FUNCTION_BLOCK TwoConCtlMulticast (* Composite Function Block Type *)
  (* Standard: 61499-2 *)
  (* Version 0.2, 2003-12-05, JHC, Rockwell Automation, Renamed from NEWCOMPFB. *)
  (* Version 0.1, 2002-01-08, JHC, Rockwell Automation, Added DLY FB as example. *)
  (* Version 0.0, 2000-05-27, JHC, Rockwell Automation *)
  (* Compiler header: package fb.rt.cs725; *)
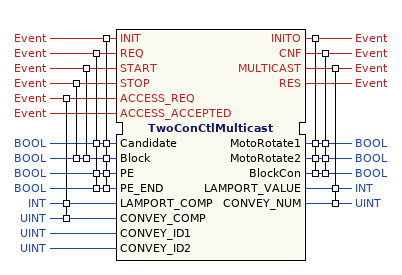
  EVENT_INPUT
    INIT WITH Candidate, Block, PE, PE_END; (* Initialization Request *)
    REQ WITH Candidate, PE, PE_END; (* Normal Execution Request *)
    START WITH Block;
    STOP WITH Block;
    ACCESS_REQ WITH LAMPORT_COMP, CONVEY_COMP;
    ACCESS_ACCEPTED;
  END_EVENT
  EVENT_OUTPUT
    INITO WITH MotoRotate1, MotoRotate2, BlockCon; (* Initialization Confirm *)
    CNF WITH MotoRotate1, MotoRotate2, BlockCon; (* Execution Confirmation *)
    MULTICAST WITH LAMPORT_VALUE, CONVEY_NUM;
    RES;
  END_EVENT
  VAR_INPUT
    Candidate : BOOL;
    Block : BOOL;
    PE : BOOL;
    PE_END : BOOL;
    LAMPORT_COMP : INT;
    CONVEY_COMP : UINT;
    CONVEY_ID1 : UINT;
    CONVEY_ID2 : UINT;
  END_VAR
  VAR_OUTPUT
    MotoRotate1 : BOOL;
    MotoRotate2 : BOOL;
    BlockCon : BOOL;
    LAMPORT_VALUE : INT;
    CONVEY_NUM : UINT;
  END_VAR
  FBS
    FC11 : ConveyorCTLMulticast(PE := 1, Block := 0, Candidate := 0);
    FC12 : ConveyorCTLMulticast;
  END_FBS
  EVENT_CONNECTIONS
    INIT TO FC11.INIT;
    REQ TO FC11.REQ;
    FC12.INITO TO INITO;
    FC12.CNF TO CNF;
    REQ TO FC12.REQ;
    STOP TO FC12.CAS_STOP;
    START TO FC12.CAS_START;
    FC12.STOP TO FC11.CAS_STOP;
    FC12.START TO FC11.CAS_START;
    FC11.INITO TO FC12.INIT;
    FC12.MULTICAST TO MULTICAST;
    FC12.RES TO RES;
    ACCESS_REQ TO FC12.ACCESS_REQ;
    ACCESS_ACCEPTED TO FC12.ACCESS_ACCEPTED;
  END_CONNECTIONS
  DATA_CONNECTIONS
    Block TO FC12.Block;
    Candidate TO FC12.Candidate;
    PE TO FC12.PE;
    FC12.BlockCon TO BlockCon;
    FC11.MotoRotate TO MotoRotate1;
    FC12.MotoRotate TO MotoRotate2;
    FC12.LAMPORT_VALUE TO LAMPORT_VALUE;
    FC12.CONVEY_NUM TO CONVEY_NUM;
    CONVEY_ID1 TO FC12.CONVEY_ID;
    CONVEY_ID2 TO FC11.CONVEY_ID;
    PE_END TO FC12.PE_END;
    LAMPORT_COMP TO FC12.LAMPORT_COMP;
    CONVEY_COMP TO FC12.CONVEY_COMP;
  END_CONNECTIONS
END_FUNCTION_BLOCK
